Staubli VAL3: POINT.dtx

public TrajPoint tTraj{}
